Staubli VAL3: CartesianTrajPt.dtx

public num nSeq
public num nPosition[3]
public num nOrientation[4]
public num nVelocity
public num nAcceleration
public num nBlendingRadius
public num nDuration
